VISUALIZATION VISU_BLANCK_MANUEL  // 1280x1024
END_VISUALIZATION

(* stored: Version 1.1.0.1, ProductVersion 3.1.4024.10
   Visu VISU_BLANCK_MANUEL: Id {9ba2baf7-1699-45bd-9972-7249f175babd} *)
